// TwinCAT 3 PLC project ScalingAndConversion
// Title: ScalingAndConversion
// Company: Beckhoff Automation LLC.
// Author: m.kleven@beckhoff.com
// ProjectVersion: 0.0.1
// Description: Scaling and conversion algorithms
// ProgramVersion: 3.1.4026.18
// project tree:
//   / E_TemperatureUnit.TcDUT, FB_LinearScaling.TcPOU, FB_TemperatureConversion.TcPOU
//   Project Information/ F_GetCompany.TcPOU, F_GetTitle.TcPOU, F_GetVersion.TcPOU
//   Version/ Global_Version.TcGVL

// ---- E_TemperatureUnit.TcDUT
{attribute 'qualified_only'}
{attribute 'strict'}
{attribute 'to_string'}
TYPE E_TemperatureUnit  :
(
   Celsius := 0,
    Fahrenheit := 1,
    Kelvin := 2,
    Rankine := 3
);
END_TYPE

// ---- Version/Global_Version.TcGVL
{attribute 'TcGenerated'}
{attribute 'no-analysis'}
{attribute 'linkalways'}
// This function has been automatically generated from the project information.
VAR_GLOBAL CONSTANT
	{attribute 'const_non_replaced'}
	stLibVersion_ScalingAndConversion : ST_LibVersion := (iMajor := 0, iMinor := 0, iBuild := 1, iRevision := 0, nFlags := 0, sVersion := '0.0.1');
END_VAR

// ---- FB_LinearScaling.TcPOU
FUNCTION_BLOCK FB_LinearScaling
VAR_INPUT
    Enable      : BOOL;          // Enable scaling
    RawValue    : LREAL;         // Raw input value (e.g., ADC counts)
    RawMin      : LREAL := 0.0;  // Minimum raw value
    RawMax      : LREAL := 4095.0; // Maximum raw value (e.g., 12-bit ADC)
    ScaledMin   : LREAL := 0.0;  // Minimum scaled value (engineering units)
    ScaledMax   : LREAL := 100.0; // Maximum scaled value (engineering units)
    LimitOutput : BOOL := TRUE;  // Limit output to scaled range
END_VAR

VAR_OUTPUT
    ScaledValue : LREAL;         // Scaled output value
    OutOfRange  : BOOL;          // Input is outside raw range
    Error       : BOOL;          // Error flag
END_VAR

VAR
    Scale       : LREAL;         // Calculated scaling factor
    Offset      : LREAL;         // Calculated offset
    TempValue   : LREAL;         // Temporary calculation value
END_VAR

IF Enable THEN
    // Input validation
    IF RawMax <= RawMin THEN
        Error := TRUE;
        ScaledValue := 0.0;
        OutOfRange := TRUE;
        RETURN;
    END_IF
    
    // Calculate scaling parameters
    Scale := (ScaledMax - ScaledMin) / (RawMax - RawMin);
    Offset := ScaledMin - (Scale * RawMin);
    
    // Check if input is within expected range
    OutOfRange := (RawValue < RawMin) OR (RawValue > RawMax);
    
    // Perform linear scaling: y = mx + b
    TempValue := Scale * RawValue + Offset;
    
    // Apply output limiting if enabled
    IF LimitOutput THEN
        IF TempValue < ScaledMin THEN
            ScaledValue := ScaledMin;
        ELSIF TempValue > ScaledMax THEN
            ScaledValue := ScaledMax;
        ELSE
            ScaledValue := TempValue;
        END_IF
    ELSE
        ScaledValue := TempValue;
    END_IF
    
    Error := FALSE;
ELSE
    ScaledValue := 0.0;
    OutOfRange := FALSE;
    Error := FALSE;
END_IF

END_FUNCTION_BLOCK

// ---- FB_TemperatureConversion.TcPOU
FUNCTION_BLOCK FB_TemperatureConversion
VAR_INPUT
    Enable       : BOOL;                                    // Enable conversion
    InputTemp    : LREAL;                                   // Input temperature value
    InputUnit    : E_TemperatureUnit := E_TemperatureUnit.Celsius;  // Input unit
    OutputUnit   : E_TemperatureUnit := E_TemperatureUnit.Fahrenheit; // Desired output unit
END_VAR

VAR_OUTPUT
    OutputTemp   : LREAL;                                   // Converted temperature
    Error        : BOOL;                                    // Error flag
    ErrorMessage : STRING(80);                              // Error description
END_VAR

VAR
    TempCelsius  : LREAL;                                   // Intermediate Celsius value
END_VAR

VAR CONSTANT
    AbsoluteZeroC : LREAL := -273.15;  // Absolute zero in Celsius
    AbsoluteZeroF : LREAL := -459.67;  // Absolute zero in Fahrenheit
END_VAR

IF Enable THEN
    Error := FALSE;
    ErrorMessage := '';
    
    // First convert input to Celsius as intermediate step
    CASE InputUnit OF
        E_TemperatureUnit.Celsius:
            TempCelsius := InputTemp;
            // Check for physically impossible temperature
            IF InputTemp < AbsoluteZeroC THEN
                Error := TRUE;
                ErrorMessage := 'Temperature below absolute zero';
                OutputTemp := 0.0;
                RETURN;
            END_IF
            
        E_TemperatureUnit.Fahrenheit:
            // Check for physically impossible temperature
            IF InputTemp < AbsoluteZeroF THEN
                Error := TRUE;
                ErrorMessage := 'Temperature below absolute zero';
                OutputTemp := 0.0;
                RETURN;
            END_IF
            TempCelsius := (InputTemp - 32.0) * 5.0 / 9.0;
            
        E_TemperatureUnit.Kelvin:
            // Check for physically impossible temperature
            IF InputTemp < 0.0 THEN
                Error := TRUE;
                ErrorMessage := 'Temperature below absolute zero';
                OutputTemp := 0.0;
                RETURN;
            END_IF
            TempCelsius := InputTemp - 273.15;
            
        E_TemperatureUnit.Rankine:
            // Check for physically impossible temperature
            IF InputTemp < 0.0 THEN
                Error := TRUE;
                ErrorMessage := 'Temperature below absolute zero';
                OutputTemp := 0.0;
                RETURN;
            END_IF
            TempCelsius := (InputTemp - 491.67) * 5.0 / 9.0;
            
        ELSE
            Error := TRUE;
            ErrorMessage := 'Invalid input temperature unit';
            OutputTemp := 0.0;
            RETURN;
    END_CASE
    
    // Now convert from Celsius to desired output unit
    CASE OutputUnit OF
        E_TemperatureUnit.Celsius:
            OutputTemp := TempCelsius;
            
        E_TemperatureUnit.Fahrenheit:
            OutputTemp := (TempCelsius * 9.0 / 5.0) + 32.0;
            
        E_TemperatureUnit.Kelvin:
            OutputTemp := TempCelsius + 273.15;
            
        E_TemperatureUnit.Rankine:
            OutputTemp := (TempCelsius + 273.15) * 9.0 / 5.0;
            
        ELSE
            Error := TRUE;
            ErrorMessage := 'Invalid output temperature unit';
            OutputTemp := 0.0;
            RETURN;
    END_CASE
    
ELSE
    OutputTemp := 0.0;
    Error := FALSE;
    ErrorMessage := '';
END_IF

END_FUNCTION_BLOCK

// ---- Project Information/F_GetCompany.TcPOU
// This function has been automatically generated from the project information.
{attribute 'signature_flag' := '1073741824'}
{attribute 'TcGenerated'}
{attribute 'no-analysis'}
FUNCTION F_GetCompany : WSTRING
VAR_INPUT
	
END_VAR

F_GetCompany := "Beckhoff Automation LLC.";

END_FUNCTION

// ---- Project Information/F_GetTitle.TcPOU
// This function has been automatically generated from the project information.
{attribute 'signature_flag' := '1073741824'}
{attribute 'TcGenerated'}
{attribute 'no-analysis'}
FUNCTION F_GetTitle : WSTRING
VAR_INPUT
	
END_VAR

F_GetTitle := "ScalingAndConversion";

END_FUNCTION

// ---- Project Information/F_GetVersion.TcPOU
// This function has been automatically generated from the project information.
{attribute 'signature_flag' := '1073741824'}
{attribute 'TcGenerated'}
{attribute 'no-analysis'}
FUNCTION F_GetVersion : ST_LibVersion
VAR_INPUT
	
END_VAR

F_GetVersion.iMajor := 0;
F_GetVersion.iMinor := 0;
F_GetVersion.iBuild := 1;
F_GetVersion.iRevision := 0;
F_GetVersion.sVersion := '0.0.1';
F_GetVersion.nFlags := 0;

END_FUNCTION
